(* IEC 61131-3 sources: vibrocore/firmware/codesys, 8 files *)

(* ---- GVL_IO.st ---- *)
(*
 * GVL_IO — Global Variable List: Physical I/O Mapping
 *
 * WAGO PFC200 XTR (750-8212) + I/O Modules:
 *   Slot 1: 750-430 XTR  — 4× Digital Input  24V DC  → %IX0.0..%IX0.3
 *   Slot 2: 750-530 XTR  — 4× Digital Output 24V DC  → %QX0.0..%QX0.3
 *   Slot 3: 750-637      — Incremental Encoder        → %IW4 (32-bit via IW4+IW5)
 *   Slot 4: 750-826      — RS-485 Modbus RTU          → COM config in hardware tree
 *   Slot 5: 750-600      — End module
 *
 * RS-485 Slave Addresses:
 *   Addr 1: Siemens V20 VFD  (Sonic Head)
 *   Addr 2: Nanotec C5-E     (Hub stepper driver)
 *)
VAR_GLOBAL

    (* =========================================================
       Slot 1 — 750-430 XTR: 4x Digital Input 24V DC
       ========================================================= *)

    (* Upper limit switch (NC wiring — FALSE = triggered) *)
    xLimitUp        AT %IX0.0 : BOOL;

    (* Lower limit switch (NC wiring — FALSE = triggered) *)
    xLimitDown      AT %IX0.1 : BOOL;

    (* Emergency stop mushroom button (NC — FALSE = pressed) *)
    xEStop_NC       AT %IX0.2 : BOOL;

    (* Hub driver alarm output (Nanotec C5-E ALM pin, active HIGH) *)
    xHubAlarm       AT %IX0.3 : BOOL;

    (* =========================================================
       Slot 2 — 750-530 XTR: 4x Digital Output 24V DC
       ========================================================= *)

    (* Spring-applied brake: HIGH = 24V energised = brake RELEASED *)
    xBrakeRelease   AT %QX0.0 : BOOL;

    (* Hub driver enable (Nanotec C5-E ENA pin, active HIGH) *)
    xHubEnable      AT %QX0.1 : BOOL;

    (* VFD fault reset pulse (momentary, 200ms) *)
    xVFD_Reset      AT %QX0.2 : BOOL;

    (* Spare digital output — reserved for alarm beacon / HMI *)
    xAlarmBeacon    AT %QX0.3 : BOOL;

    (* =========================================================
       Slot 3 — 750-637: Incremental Encoder
       Encoder on hub chain shaft (1000 ppr, quadrature)
       Mapped as 32-bit signed integer (IW4 = low word, IW5 = high word)
       ========================================================= *)

    iEncoderLow     AT %IW4   : INT;
    iEncoderHigh    AT %IW5   : INT;

END_VAR

(* ---- GVL_PARAMS.st ---- *)
(*
 * GVL_PARAMS — Machine Parameters and Constants
 *
 * All physical machine constants. Verify against actual hardware
 * before commissioning. Speeds and thresholds are starting values
 * for field calibration.
 *)
VAR_GLOBAL CONSTANT

    (* =========================================================
       Hub Kinematics
       NEMA 42 + Neugart PLPE120-040 (40:1) + 10B-2 chain + 15T sprocket
       ========================================================= *)

    (* Encoder pulses per mm of carriage travel
       = (pulses/rev × gear_ratio) / (sprocket_teeth × chain_pitch)
       = (1000 × 4 × 40) / (15 × 15.875) = 160000 / 238.125 ≈ 671.9 *)
    rENCODER_PULSES_PER_MM  : REAL := 671.9;

    (* Maximum carriage travel (mm) — physical mast stroke *)
    rMAX_STROKE_MM          : REAL := 1300.0;

    (* Default sampling target depth (mm from home) *)
    rTARGET_DEPTH_MM        : REAL := 1200.0;

    (* Hub speed setpoints (mm/s) *)
    rSPEED_PENETRATE_MMS    : REAL := 15.0;   (* push-in with sonic active *)
    rSPEED_RETRACT_MMS      : REAL := 50.0;   (* pull-out after sonic stop *)
    rSPEED_MANUAL_MMS       : REAL := 30.0;   (* manual jog speed *)
    rSPEED_HOMING_MMS       : REAL := 40.0;   (* homing to upper limit *)

    (* Position tolerance for "at target" check (mm) *)
    rPOS_TOLERANCE_MM       : REAL := 5.0;

    (* =========================================================
       Hub Modbus (Nanotec C5-E — CiA 402 via Modbus RTU)
       ========================================================= *)

    iHUB_SLAVE_ADDR         : INT  := 2;

    (* Modbus register addresses (holding registers, 0-based Modbus) *)
    iHUB_REG_CONTROLWORD    : INT  := 16#6040;  (* CiA 402 control word *)
    iHUB_REG_STATUSWORD     : INT  := 16#6041;  (* CiA 402 status word *)
    iHUB_REG_TARGET_VEL     : INT  := 16#60FF;  (* target velocity, rpm *)
    iHUB_REG_ACTUAL_POS     : INT  := 16#6064;  (* position actual, encoder counts *)
    iHUB_REG_OPMODE         : INT  := 16#6060;  (* modes of operation: 3=Velocity *)

    (* CiA 402 control words *)
    wHUB_CW_SHUTDOWN        : WORD := 16#0006;  (* Shutdown *)
    wHUB_CW_ENABLE          : WORD := 16#000F;  (* Switch On + Enable Op *)
    wHUB_CW_QUICKSTOP       : WORD := 16#000B;  (* Quick stop *)
    wHUB_CW_FAULT_RESET     : WORD := 16#0080;  (* Fault reset *)

    (* =========================================================
       VFD Modbus (Siemens V20 — USS/Modbus profile)
       Standard parameter channel + process data (PKW + PZD)
       ========================================================= *)

    iVFD_SLAVE_ADDR         : INT  := 1;

    (* Process data input/output word addresses (0-based) *)
    iVFD_REG_CONTROL        : INT  := 100;   (* STW1: control word *)
    iVFD_REG_FREQ_SP        : INT  := 101;   (* HSW: freq setpoint ×100 Hz *)
    iVFD_REG_STATUS         : INT  := 110;   (* ZSW1: status word *)
    iVFD_REG_FREQ_ACT       : INT  := 111;   (* HIW: actual frequency ×100 Hz *)
    iVFD_REG_CURRENT        : INT  := 112;   (* actual current ×10 A *)

    (* V20 STW1 control words *)
    wVFD_CW_START           : WORD := 16#047F;  (* bits: ON + no OFF2 + no OFF3 + OpEnable *)
    wVFD_CW_STOP_NORMAL     : WORD := 16#047E;  (* OFF1: ramp down via P1121 *)
    wVFD_CW_STOP_FAST       : WORD := 16#047B;  (* OFF3: fast ramp via P1135 + DC brake *)
    wVFD_CW_FAULT_RESET     : WORD := 16#04FE;  (* fault acknowledgement *)

    (* Frequency limits (Hz) *)
    rVFD_FREQ_MIN_HZ        : REAL := 30.0;
    rVFD_FREQ_MAX_HZ        : REAL := 110.0;
    rVFD_FREQ_DEFAULT_HZ    : REAL := 100.0;

    (* Ramp rates for software-side tracking (Hz per 100ms cycle) *)
    rVFD_RAMP_UP_HZ_STEP    : REAL := 1.5;   (* ≈15 Hz/s -->  ~7s to 100 Hz *)
    rVFD_RAMP_DN_HZ_STEP    : REAL := 4.5;   (* ≈45 Hz/s --> normal stop *)

    (* Skip resonance band: avoid 8–25 Hz during run-up *)
    rVFD_SKIP_BAND_LOW_HZ   : REAL := 8.0;
    rVFD_SKIP_BAND_HIGH_HZ  : REAL := 25.0;

    (* =========================================================
       Safety / Stone Detection
       ========================================================= *)

    (* VFD output current threshold for stone detection (% of motor rated) *)
    rSTONE_CURRENT_PCT_THR  : REAL := 130.0;

    (* Debounce time before stone alarm is confirmed *)
    tSTONE_DEBOUNCE         : TIME := T#250MS;

    (* Hub retract distance after stone detection (mm) *)
    rSTONE_RETRACT_MM       : REAL := 50.0;

    (* Max wait time for Sonic head to confirm stop before fault *)
    tSONIC_STOP_TIMEOUT     : TIME := T#5S;

    (* =========================================================
       Data / Identity
       ========================================================= *)

    sMACHINE_ID             : STRING[20] := 'VIBROCORE-001';
    sHARDWARE_VERSION       : STRING[10] := 'V1.0';
    sFIRMWARE_VERSION       : STRING[10] := '1.0.0';

END_VAR

(* ---- FB_DataLogger.st ---- *)
(*
 * FB_DataLogger — Cycle Data Logging and MQTT Payload Builder
 *
 * On each completed sampling cycle, assembles a JSON payload containing:
 *   - Machine ID, cycle number, timestamp
 *   - GPS coordinates (received from SE050/ESP32-C3 via UART → Modbus)
 *   - Achieved depth, VFD frequency, motor current
 *   - sign_pending flag → ESP32-C3 picks this up and signs via SE050 (secp256k1)
 *     then publishes to RDDL/Planetmint for VM0042 data provenance
 *
 * UART connection ESP32-C3 (RDDL Trust Wallet):
 *   WAGO COM1 (750-650 or PFC onboard UART) ↔ ESP32-C3 TX/RX
 *   Protocol: simple JSON lines at 115200 baud
 *   ESP32-C3 pushes GPS fixes every 1s: {"lat":47.123,"lon":16.456,"fix":"RTK"}
 *   WAGO sends completed cycle JSON: {"machine_id":...,"sign_pending":true}
 *   ESP32-C3 signs with SE050 and forwards to RDDL
 *
 * MQTT (WAGO onboard MQTT client via e!COCKPIT or Node-RED on PFC Linux):
 *   Topic: vibrocore/{machine_id}/cycles
 *   Broker: configured in WAGO web interface (wago-mqtt-config)
 *)
FUNCTION_BLOCK FB_DataLogger
VAR_INPUT
    xCycleTrigger       : BOOL;   (* rising edge = new cycle to log *)
    rDepth_mm           : REAL;
    rFreq_Hz            : REAL;
    rCurrent_A          : REAL;
    iSafetyReason       : INT;    (* 0=normal, >0 = what caused stop *)
END_VAR

VAR_OUTPUT
    sJSON_Payload       : STRING[500];
    xNewPayload         : BOOL;   (* TRUE for one PLC cycle when payload ready *)
    iCycleCount         : INT;
END_VAR

VAR
    (* GPS data received from ESP32-C3 — updated via UART parse task *)
    rGPS_Lat            : REAL := 0.0;
    rGPS_Lon            : REAL := 0.0;
    sGPS_Fix            : STRING[10] := 'NONE';

    tTimestamp          : TON;   (* simple uptime counter in seconds *)
    iUptimeSec          : DINT  := 0;

    xTriggerEdge        : R_TRIG;
    xPayloadSent        : BOOL;
END_VAR

(* ---- Uptime counter ---- *)
tTimestamp(IN := TRUE, PT := T#1S);
IF tTimestamp.Q THEN
    tTimestamp(IN := FALSE);
    iUptimeSec := iUptimeSec + 1;
END_IF;

(* ---- Rising edge on cycle trigger ---- *)
xTriggerEdge(CLK := xCycleTrigger);
xNewPayload := FALSE;

IF xTriggerEdge.Q THEN
    iCycleCount := iCycleCount + 1;

    (*
     * Build JSON payload manually (no dynamic allocator in IEC 61131-3).
     * Payload is read by the ESP32-C3 on COM1. The ESP32-C3 appends the
     * SE050 secp256k1 signature and publishes to RDDL/Planetmint.
     *
     * Example output:
     * {"machine_id":"VIBROCORE-001","fw":"1.0.0","cycle":1,
     *  "uptime_s":3600,"depth_mm":1198.4,"freq_hz":100.0,
     *  "current_a":1.38,"stop_reason":0,
     *  "lat":47.1234567,"lon":16.4567890,"fix":"RTK",
     *  "sign_pending":true}
     *)
    sJSON_Payload := CONCAT('{"machine_id":"',
                     CONCAT(GVL_PARAMS.sMACHINE_ID,         '","'));
    sJSON_Payload := CONCAT(sJSON_Payload,
                     CONCAT('fw":"',
                     CONCAT(GVL_PARAMS.sFIRMWARE_VERSION,   '",')));
    sJSON_Payload := CONCAT(sJSON_Payload,
                     CONCAT('"cycle":',
                     CONCAT(INT_TO_STRING(iCycleCount),     ',')));
    sJSON_Payload := CONCAT(sJSON_Payload,
                     CONCAT('"uptime_s":',
                     CONCAT(DINT_TO_STRING(iUptimeSec),     ',')));
    sJSON_Payload := CONCAT(sJSON_Payload,
                     CONCAT('"depth_mm":',
                     CONCAT(REAL_TO_STRING(rDepth_mm),      ',')));
    sJSON_Payload := CONCAT(sJSON_Payload,
                     CONCAT('"freq_hz":',
                     CONCAT(REAL_TO_STRING(rFreq_Hz),       ',')));
    sJSON_Payload := CONCAT(sJSON_Payload,
                     CONCAT('"current_a":',
                     CONCAT(REAL_TO_STRING(rCurrent_A),     ',')));
    sJSON_Payload := CONCAT(sJSON_Payload,
                     CONCAT('"stop_reason":',
                     CONCAT(INT_TO_STRING(iSafetyReason),   ',')));
    sJSON_Payload := CONCAT(sJSON_Payload,
                     CONCAT('"lat":',
                     CONCAT(REAL_TO_STRING(rGPS_Lat),       ',')));
    sJSON_Payload := CONCAT(sJSON_Payload,
                     CONCAT('"lon":',
                     CONCAT(REAL_TO_STRING(rGPS_Lon),       ',')));
    sJSON_Payload := CONCAT(sJSON_Payload,
                     CONCAT('"fix":"',
                     CONCAT(sGPS_Fix,                       '",')));
    sJSON_Payload := CONCAT(sJSON_Payload, '"sign_pending":true}');

    xNewPayload := TRUE;
END_IF;

(* ---- FB_HubControl.st ---- *)
(*
 * FB_HubControl — Hub Lift/Lower State Machine
 *
 * Controls NEMA 42 stepper via Nanotec C5-E (Modbus RTU, CiA 402).
 * Drive train: NEMA42 → Neugart PLPE120-040 (40:1) → 10B-2 chain → carriage.
 *
 * CRITICAL INTERLOCK:
 *   Hub may ONLY move upward (retract) when xSonicConfirmedStopped = TRUE.
 *   This prevents soil sample falling out during extraction.
 *   Stone detection also requires sonic stop FIRST — never retract while vibrating.
 *
 * State machine:
 *   0 IDLE          — brake engaged, motor disabled
 *   1 HOMING        — move up until xLimitUp (establishes position zero)
 *   2 DRILL_WAIT    — waiting for sonic confirmed running before hub moves
 *   3 DRILLING      — hub moves down at penetration speed
 *   4 STOP_SONIC    — target/stone reached: brake hub, request sonic fast-stop
 *   5 RETRACT       — sonic confirmed stopped, hub moves up
 *   6 ESTOP_HOLD    — emergency stop: brake engaged, waiting for release
 *   7 FAULT         — driver alarm or timeout
 *)
FUNCTION_BLOCK FB_HubControl
VAR_INPUT
    xEnable                 : BOOL;
    xSafeState              : BOOL;   (* from FB_Safety: freeze all motion *)
    xStoneDetected          : BOOL;   (* from FB_Safety: obstacle detected *)
    xSonicRunning           : BOOL;   (* from FB_SonicHead: motors spinning *)
    xSonicConfirmedStopped  : BOOL;   (* from FB_SonicHead: motors confirmed at rest *)

    rTargetDepth_mm         : REAL;   (* sampling target depth (mm from home) *)

    (* Manual jog inputs (active only in IDLE state) *)
    xCmdJogDown             : BOOL;
    xCmdJogUp               : BOOL;

    (* Auto cycle start *)
    xCmdCycleStart          : BOOL;

    (* Fault reset *)
    xCmdReset               : BOOL;
END_VAR

VAR_OUTPUT
    rPosition_mm        : REAL;    (* current carriage position from home, mm *)
    xAtHome             : BOOL;    (* carriage at upper limit *)
    xAtTarget           : BOOL;    (* carriage within tolerance of target depth *)
    xNeedSonicStop      : BOOL;    (* TRUE = request sonic fast-stop *)
    xCycleComplete      : BOOL;    (* pulse: TRUE for one cycle after retract done *)
    xFault              : BOOL;
    eState              : INT;

    (* Physical outputs — mapped by PRG_Main to GVL_IO *)
    xBrakeRelease_out   : BOOL;
    xHubEnable_out      : BOOL;
END_VAR

VAR
    (* Modbus to Nanotec C5-E *)
    fbMBWrite           : WagoModbusMasterRtu.MB_RTU_WRITE_REGS;
    fbMBRead            : WagoModbusMasterRtu.MB_RTU_READ_REGS;
    awWriteRegs         : ARRAY[0..1] OF WORD;   (* controlword + target velocity *)
    awReadRegs          : ARRAY[0..2] OF WORD;   (* statusword + actual pos low/high *)

    tMBCycle            : TON;
    tSonicStopTimeout   : TON;
    tCyclePulse         : TON;

    iSpeedSetpoint_rpm  : INT;   (* speed sent to C5-E, signed: + = down, - = up *)
    wHubCtrlWord        : WORD;

    (* 32-bit encoder position from Modbus *)
    lActualPos          : LINT;
    iPosPrev            : INT;
END_VAR

(* ---- Position calculation (encoder → mm) ---- *)
(* Combine low and high words from C5-E position register *)
lActualPos   := SHL(LINT#0 + INT_TO_LINT(awReadRegs[2]), 16)
                + INT_TO_LINT(WORD_TO_INT(awReadRegs[1]));
rPosition_mm := LINT_TO_REAL(lActualPos) / GVL_PARAMS.rENCODER_PULSES_PER_MM;

(* ---- Derived position flags ---- *)
xAtHome   := NOT GVL_IO.xLimitUp_NC;   (* NC: FALSE = triggered = home *)
xAtTarget := (rPosition_mm >= rTargetDepth_mm - GVL_PARAMS.rPOS_TOLERANCE_MM)
          AND (rPosition_mm <= rTargetDepth_mm + GVL_PARAMS.rPOS_TOLERANCE_MM);

(* ---- Global E-Stop / Safety override ---- *)
IF xSafeState AND eState <> 6 AND eState <> 7 THEN
    wHubCtrlWord        := GVL_PARAMS.wHUB_CW_QUICKSTOP;
    iSpeedSetpoint_rpm  := 0;
    xBrakeRelease_out   := FALSE;   (* brake engages *)
    xHubEnable_out      := FALSE;
    xNeedSonicStop      := TRUE;
    eState              := 6;
END_IF;

(* ---- State machine ---- *)
CASE eState OF

    (* ============================================================ *)
    0: (* IDLE *)
    (* ============================================================ *)
        wHubCtrlWord       := GVL_PARAMS.wHUB_CW_SHUTDOWN;
        iSpeedSetpoint_rpm := 0;
        xBrakeRelease_out  := FALSE;
        xHubEnable_out     := FALSE;
        xNeedSonicStop     := FALSE;
        xFault             := FALSE;
        xCyclePulse(IN := FALSE);

        IF xCmdCycleStart AND xEnable AND NOT xSafeState THEN
            eState := 1;   (* Home first, then drill *)
        ELSIF xCmdJogDown AND xEnable AND NOT GVL_IO.xLimitDown AND NOT xSafeState THEN
            xBrakeRelease_out  := TRUE;
            xHubEnable_out     := TRUE;
            wHubCtrlWord       := GVL_PARAMS.wHUB_CW_ENABLE;
            iSpeedSetpoint_rpm := REAL_TO_INT(GVL_PARAMS.rSPEED_MANUAL_MMS
                                              * GVL_PARAMS.rENCODER_PULSES_PER_MM / 1000.0 * 60.0);
        ELSIF xCmdJogUp AND xEnable AND NOT GVL_IO.xLimitUp AND NOT xSafeState THEN
            xBrakeRelease_out  := TRUE;
            xHubEnable_out     := TRUE;
            wHubCtrlWord       := GVL_PARAMS.wHUB_CW_ENABLE;
            iSpeedSetpoint_rpm := -REAL_TO_INT(GVL_PARAMS.rSPEED_MANUAL_MMS
                                               * GVL_PARAMS.rENCODER_PULSES_PER_MM / 1000.0 * 60.0);
        END_IF;

    (* ============================================================ *)
    1: (* HOMING — move up to upper limit switch *)
    (* ============================================================ *)
        xBrakeRelease_out  := TRUE;
        xHubEnable_out     := TRUE;
        wHubCtrlWord       := GVL_PARAMS.wHUB_CW_ENABLE;
        iSpeedSetpoint_rpm := -REAL_TO_INT(GVL_PARAMS.rSPEED_HOMING_MMS
                                           * GVL_PARAMS.rENCODER_PULSES_PER_MM / 1000.0 * 60.0);

        IF xAtHome THEN
            (* Limit reached — stop motor, set position origin in C5-E *)
            wHubCtrlWord       := GVL_PARAMS.wHUB_CW_SHUTDOWN;
            iSpeedSetpoint_rpm := 0;
            xBrakeRelease_out  := FALSE;
            xHubEnable_out     := FALSE;
            eState             := 2;   (* → wait for sonic *)
        END_IF;

    (* ============================================================ *)
    2: (* DRILL_WAIT — wait for sonic confirmed running *)
    (* ============================================================ *)
        xBrakeRelease_out  := FALSE;
        xHubEnable_out     := FALSE;
        iSpeedSetpoint_rpm := 0;

        IF xSonicRunning THEN
            eState := 3;
        END_IF;

        IF NOT xEnable OR xSafeState THEN
            eState := 0;
        END_IF;

    (* ============================================================ *)
    3: (* DRILLING — hub moves down, sonic running *)
    (* ============================================================ *)
        xBrakeRelease_out  := TRUE;
        xHubEnable_out     := TRUE;
        wHubCtrlWord       := GVL_PARAMS.wHUB_CW_ENABLE;
        iSpeedSetpoint_rpm := REAL_TO_INT(GVL_PARAMS.rSPEED_PENETRATE_MMS
                                          * GVL_PARAMS.rENCODER_PULSES_PER_MM / 1000.0 * 60.0);

        (* Stop drilling on target OR stone *)
        IF xAtTarget OR xStoneDetected OR GVL_IO.xLimitDown THEN
            (* Engage brake, request sonic fast-stop *)
            wHubCtrlWord       := GVL_PARAMS.wHUB_CW_QUICKSTOP;
            iSpeedSetpoint_rpm := 0;
            xBrakeRelease_out  := FALSE;
            xHubEnable_out     := FALSE;
            xNeedSonicStop     := TRUE;
            eState             := 4;
        END_IF;

    (* ============================================================ *)
    4: (* STOP_SONIC — brake engaged, waiting for sonic to confirm stop *)
    (* Hub MUST NOT move. Retract only after xSonicConfirmedStopped. *)
    (* ============================================================ *)
        xBrakeRelease_out  := FALSE;
        xHubEnable_out     := FALSE;
        iSpeedSetpoint_rpm := 0;
        xNeedSonicStop     := TRUE;   (* keep requesting fast stop *)

        tSonicStopTimeout(
            IN := TRUE,
            PT := GVL_PARAMS.tSONIC_STOP_TIMEOUT
        );

        IF xSonicConfirmedStopped THEN
            tSonicStopTimeout(IN := FALSE);
            xNeedSonicStop := FALSE;
            eState := 5;   (* → now safe to retract *)
        END_IF;

        IF tSonicStopTimeout.Q THEN
            tSonicStopTimeout(IN := FALSE);
            xFault := TRUE;
            eState := 7;   (* timeout waiting for sonic → fault *)
        END_IF;

    (* ============================================================ *)
    5: (* RETRACT — sonic confirmed stopped, hub moves up *)
    (* ============================================================ *)
        xBrakeRelease_out  := TRUE;
        xHubEnable_out     := TRUE;
        wHubCtrlWord       := GVL_PARAMS.wHUB_CW_ENABLE;
        iSpeedSetpoint_rpm := -REAL_TO_INT(GVL_PARAMS.rSPEED_RETRACT_MMS
                                           * GVL_PARAMS.rENCODER_PULSES_PER_MM / 1000.0 * 60.0);

        IF xAtHome THEN
            wHubCtrlWord       := GVL_PARAMS.wHUB_CW_SHUTDOWN;
            iSpeedSetpoint_rpm := 0;
            xBrakeRelease_out  := FALSE;
            xHubEnable_out     := FALSE;
            (* Pulse xCycleComplete for one cycle *)
            tCyclePulse(IN := TRUE, PT := T#500MS);
            xCycleComplete     := tCyclePulse.Q;
            IF tCyclePulse.Q THEN
                tCyclePulse(IN := FALSE);
                xCycleComplete := FALSE;
                eState := 0;
            END_IF;
        END_IF;

    (* ============================================================ *)
    6: (* ESTOP_HOLD — hold until E-Stop released and reset *)
    (* ============================================================ *)
        wHubCtrlWord       := GVL_PARAMS.wHUB_CW_QUICKSTOP;
        iSpeedSetpoint_rpm := 0;
        xBrakeRelease_out  := FALSE;
        xHubEnable_out     := FALSE;
        xNeedSonicStop     := TRUE;

        IF NOT xSafeState AND xCmdReset THEN
            xNeedSonicStop := FALSE;
            eState := 1;   (* Re-home after E-Stop *)
        END_IF;

    (* ============================================================ *)
    7: (* FAULT — driver alarm or sonic stop timeout *)
    (* ============================================================ *)
        wHubCtrlWord       := GVL_PARAMS.wHUB_CW_QUICKSTOP;
        iSpeedSetpoint_rpm := 0;
        xBrakeRelease_out  := FALSE;
        xHubEnable_out     := FALSE;
        xFault             := TRUE;

        IF xCmdReset AND NOT xSafeState AND NOT GVL_IO.xHubAlarm THEN
            xFault := FALSE;
            eState := 0;
        END_IF;

END_CASE;

(* ---- Nanotec C5-E Modbus write (20ms cycle) ---- *)
tMBCycle(IN := NOT tMBCycle.Q, PT := T#20MS);
IF tMBCycle.Q THEN
    awWriteRegs[0] := wHubCtrlWord;
    awWriteRegs[1] := INT_TO_WORD(iSpeedSetpoint_rpm);

    fbMBWrite(
        bExecute      := TRUE,
        nSlaveAddress := BYTE#2,
        eFunction     := WagoModbusMasterRtu.eMBFC.WriteMultipleRegisters,
        nStartAddress := INT_TO_WORD(GVL_PARAMS.iHUB_REG_CONTROLWORD),
        nQuantity     := 2,
        pData         := ADR(awWriteRegs),
        nDataLen      := SIZEOF(awWriteRegs)
    );

    fbMBRead(
        bExecute      := TRUE,
        nSlaveAddress := BYTE#2,
        eFunction     := WagoModbusMasterRtu.eMBFC.ReadHoldingRegisters,
        nStartAddress := INT_TO_WORD(GVL_PARAMS.iHUB_REG_STATUSWORD),
        nQuantity     := 3,
        pData         := ADR(awReadRegs),
        nDataLen      := SIZEOF(awReadRegs)
    );
END_IF;

(* ---- FB_ModbusVFD.st ---- *)
(*
 * FB_ModbusVFD — Siemens V20 VFD Communication via Modbus RTU
 *
 * Hardware: WAGO 750-826 RS-485 module, COM2 port
 * VFD: Siemens SINAMICS V20, Modbus slave address 1
 *
 * V20 pre-commissioning (set via BOP or STARTER):
 *   P0700 = 5     (command source: Modbus)
 *   P1000 = 5     (freq setpoint: Modbus)
 *   P2010[0] = 6  (Modbus baud: 9600)
 *   P2011[0] = 1  (slave address: 1)
 *   P2012[0] = 2  (PZD word count: 2)
 *   P1120 = 5.0   (ramp-up time, s)
 *   P1121 = 3.0   (ramp-down time OFF1, s)
 *   P1135 = 0.3   (ramp-down time OFF3 fast-stop, s)
 *   P1232 = 100   (DC braking current %)
 *   P1233 = 0.5   (DC braking duration, s)
 *
 * Control word bits (STW1):
 *   Bit 0: ON/OFF1  (0 = ramp to stop via P1121)
 *   Bit 1: no OFF2  (0 = coast to stop — keep 1)
 *   Bit 2: no OFF3  (0 = fast stop via P1135 — used for fast stop)
 *   Bit 3: enable operation
 *   Bit 6: setpoint enable
 *   Bit 7: fault acknowledge
 *
 * Note: Modbus library used is WagoAppModbusMasterRtu (WAGO CODESYS package).
 * Import via Library Manager: WagoAppModbusMasterRtu >= 1.1.0.0
 *)
FUNCTION_BLOCK FB_ModbusVFD
VAR_INPUT
    xEnable         : BOOL;   (* FALSE = VFD disabled, no communication *)
    xStart          : BOOL;   (* TRUE = run motor *)
    xFastStop       : BOOL;   (* TRUE = OFF3 immediately (stone / safety) *)
    xFaultReset     : BOOL;   (* rising edge = reset VFD fault *)
    rFreqSetpoint   : REAL;   (* Hz, clamped internally to MIN/MAX *)
END_VAR

VAR_OUTPUT
    xRunning        : BOOL;   (* TRUE = VFD reports motor running *)
    xReady          : BOOL;   (* TRUE = VFD ready for start command *)
    xFault          : BOOL;   (* TRUE = VFD in fault state *)
    rFreqActual     : REAL;   (* Hz — actual output frequency *)
    rCurrentActual  : REAL;   (* A  — actual output current *)
    rCurrent_pct    : REAL;   (* % of motor rated current (rated = 1.45A) *)
    xCommError      : BOOL;   (* TRUE = Modbus communication lost *)
END_VAR

VAR
    (* Modbus master FB — WagoAppModbusMasterRtu library *)
    fbMBWrite       : WagoModbusMasterRtu.MB_RTU_WRITE_REGS;
    fbMBRead        : WagoModbusMasterRtu.MB_RTU_READ_REGS;

    awWriteRegs     : ARRAY[0..1] OF WORD;   (* control + freq setpoint *)
    awReadRegs      : ARRAY[0..2] OF WORD;   (* status + freq actual + current *)

    wControlWord    : WORD;
    iFreqRaw        : INT;

    tCycle          : TON;     (* 20ms poll cycle *)
    tCommTimeout    : TON;     (* Modbus comms watchdog *)

    xResetEdge      : R_TRIG;
    xLastFaultReset : BOOL;

    (* Motor rated current for % calculation — OLI MVE 400/6-HF: 1.45A at 230V 3ph *)
    rRATED_CURRENT  : REAL := 1.45;
END_VAR

(* ---- Fault reset edge detection ---- *)
xResetEdge(CLK := xFaultReset);

(* ---- Build control word ---- *)
IF NOT xEnable THEN
    wControlWord := 16#0000;   (* fully disabled *)

ELSIF xFastStop THEN
    (* OFF3: bit 2 = 0 → VFD uses P1135 ramp + DC brake *)
    (* Achieves motor stop in ~200–400ms (vs 3+ s for normal ramp) *)
    wControlWord := GVL_PARAMS.wVFD_CW_STOP_FAST;

ELSIF xResetEdge.Q THEN
    wControlWord := GVL_PARAMS.wVFD_CW_FAULT_RESET;

ELSIF xStart THEN
    wControlWord := GVL_PARAMS.wVFD_CW_START;

ELSE
    (* Normal stop: OFF1, ramps down via P1121 *)
    wControlWord := GVL_PARAMS.wVFD_CW_STOP_NORMAL;
END_IF;

(* ---- Frequency setpoint (V20: value = Hz × 100) ---- *)
iFreqRaw := REAL_TO_INT(
    MAX(GVL_PARAMS.rVFD_FREQ_MIN_HZ,
        MIN(GVL_PARAMS.rVFD_FREQ_MAX_HZ, rFreqSetpoint)) * 100.0
);

(* ---- Pack write registers ---- *)
awWriteRegs[0] := wControlWord;
awWriteRegs[1] := INT_TO_WORD(iFreqRaw);

(* ---- 20ms poll cycle ---- *)
tCycle(IN := NOT tCycle.Q, PT := T#20MS);

IF tCycle.Q AND xEnable THEN

    (* Write: control word + freq setpoint *)
    fbMBWrite(
        bExecute     := TRUE,
        nSlaveAddress := BYTE#1,
        eFunction    := WagoModbusMasterRtu.eMBFC.WriteMultipleRegisters,
        nStartAddress := INT_TO_WORD(GVL_PARAMS.iVFD_REG_CONTROL),
        nQuantity    := 2,
        pData        := ADR(awWriteRegs),
        nDataLen     := SIZEOF(awWriteRegs)
    );

    (* Read: status word + actual freq + actual current *)
    fbMBRead(
        bExecute     := TRUE,
        nSlaveAddress := BYTE#1,
        eFunction    := WagoModbusMasterRtu.eMBFC.ReadHoldingRegisters,
        nStartAddress := INT_TO_WORD(GVL_PARAMS.iVFD_REG_STATUS),
        nQuantity    := 3,
        pData        := ADR(awReadRegs),
        nDataLen     := SIZEOF(awReadRegs)
    );

    IF fbMBRead.bDone AND NOT fbMBRead.bError THEN
        xCommError  := FALSE;
        (* ZSW1 status word bits *)
        xReady      := awReadRegs[0].1;   (* Bit 1: ready to switch on *)
        xRunning    := awReadRegs[0].2;   (* Bit 2: operation enabled / running *)
        xFault      := awReadRegs[0].3;   (* Bit 3: fault *)
        rFreqActual := WORD_TO_INT(awReadRegs[1]) / 100.0;
        rCurrentActual := WORD_TO_INT(awReadRegs[2]) / 10.0;
        rCurrent_pct   := (rCurrentActual / rRATED_CURRENT) * 100.0;
        tCommTimeout(IN := FALSE);
    ELSE
        tCommTimeout(IN := TRUE, PT := T#2S);
        xCommError := tCommTimeout.Q;
    END_IF;

END_IF;

(* ---- FB_Safety.st ---- *)
(*
 * FB_Safety — Safety Monitor Function Block
 *
 * Evaluates all safety-relevant inputs and sets xSafeState.
 * When xSafeState = TRUE, all motion must stop immediately.
 *
 * Safety categories addressed:
 *   - E-Stop: Category 3 (redundant NC wiring evaluated here)
 *   - Limit switches: NC wiring, software evaluation
 *   - Overcurrent / stone detection: software function
 *   - Hub driver fault: hardware alarm signal
 *   - VFD fault: reported by FB_ModbusVFD
 *
 * IMPORTANT: This FB does NOT directly cut power. Physical power cut
 * is handled by the safety relay (Pilz PNOZ or equivalent) wired in
 * series with the 24V supply to the VFD enable and brake circuit.
 * This FB provides the software-level interlock for the state machines.
 *)
FUNCTION_BLOCK FB_Safety
VAR_INPUT
    (* E-Stop NC contact — FALSE when button pressed *)
    xEStop_NC           : BOOL;

    (* Limit switches — NC wiring, FALSE = triggered *)
    xLimitUp_NC         : BOOL;
    xLimitDown_NC       : BOOL;

    (* Hub driver alarm output (active HIGH) *)
    xHubAlarm           : BOOL;

    (* VFD fault flag from FB_ModbusVFD *)
    xVFD_Fault          : BOOL;

    (* VFD output current as percentage of motor rated current
       Provided by FB_ModbusVFD after scaling *)
    rVFD_Current_pct    : REAL;

    (* Current hub movement direction (TRUE = moving down) *)
    xHubMovingDown      : BOOL;

    (* Current hub movement direction (TRUE = moving up) *)
    xHubMovingUp        : BOOL;
END_VAR

VAR_OUTPUT
    (* TRUE = safe state active — all motion must stop *)
    xSafeState          : BOOL;

    (* TRUE = stone/obstacle detected during penetration *)
    xStoneDetected      : BOOL;

    (* Upper limit triggered (only blocks upward movement) *)
    xLimitUpTriggered   : BOOL;

    (* Lower limit triggered (only blocks downward movement) *)
    xLimitDownTriggered : BOOL;

    (* Reason code: 0=OK 1=EStop 2=HubAlarm 3=VFD 4=Stone *)
    eSafetyReason       : INT;
END_VAR

VAR
    tStoneDebounce      : TON;
END_VAR

(* ---- Limit switch evaluation (NC contacts: FALSE = triggered) ---- *)
xLimitUpTriggered   := NOT xLimitUp_NC;
xLimitDownTriggered := NOT xLimitDown_NC;

(* ---- Stone detection with debounce ---- *)
tStoneDebounce(
    IN := rVFD_Current_pct > GVL_PARAMS.rSTONE_CURRENT_PCT_THR,
    PT := GVL_PARAMS.tSTONE_DEBOUNCE
);
xStoneDetected := tStoneDebounce.Q;

(* ---- Safe state evaluation (priority order) ---- *)
xSafeState    := FALSE;
eSafetyReason := 0;

IF NOT xEStop_NC THEN
    (* E-Stop has highest priority — hard stop *)
    xSafeState    := TRUE;
    eSafetyReason := 1;

ELSIF xHubAlarm THEN
    (* Hub driver hardware fault *)
    xSafeState    := TRUE;
    eSafetyReason := 2;

ELSIF xVFD_Fault THEN
    (* VFD hardware fault *)
    xSafeState    := TRUE;
    eSafetyReason := 3;

ELSIF xStoneDetected THEN
    (* Overcurrent → stone/obstacle — handled by state machine,
       but also sets safe state to freeze motion *)
    xSafeState    := TRUE;
    eSafetyReason := 4;

ELSIF xLimitUpTriggered AND xHubMovingUp THEN
    (* Limit in direction of travel — stop motion *)
    xSafeState    := TRUE;
    eSafetyReason := 5;

ELSIF xLimitDownTriggered AND xHubMovingDown THEN
    (* Limit in direction of travel — stop motion *)
    xSafeState    := TRUE;
    eSafetyReason := 6;
END_IF;

(* ---- FB_SonicHead.st ---- *)
(*
 * FB_SonicHead — Sonic Head State Machine
 *
 * Controls 2× OLI MVE 400/6-HF via Siemens V20 VFD (Modbus RTU).
 * Provides adaptive frequency control based on VFD load current.
 *
 * CRITICAL STOP BEHAVIOUR:
 *   - xFastStop = TRUE  → OFF3 command to VFD immediately
 *                         VFD uses P1135 ramp (0.3s) + DC injection braking
 *                         Expected motor standstill: 200–400ms
 *   - xFastStop = FALSE → OFF1 normal ramp (P1121, 3s) for end-of-cycle stop
 *
 * State machine:
 *   0 IDLE       — VFD disabled, motors at rest
 *   1 STARTING   — VFD enabled, ramping up, skip resonance band
 *   2 RUNNING    — Full speed, adaptive freq control active
 *   3 STOPPING   — Normal OFF1 stop (end of cycle)
 *   4 FAST_STOP  — OFF3 stop (stone / safety / E-Stop)
 *   5 FAULT      — VFD or comms fault, waits for reset
 *
 * Output xConfirmedStopped = TRUE only when VFD reports NOT running
 * AND state machine is in IDLE. Hub retract must wait for this.
 *)
FUNCTION_BLOCK FB_SonicHead
VAR_INPUT
    xEnable         : BOOL;   (* Allow sonic head to run *)
    xSafeState      : BOOL;   (* Safety FB active → fast stop *)
    xFastStop       : BOOL;   (* External fast stop request (stone, end-of-cycle) *)
    rTargetFreq_Hz  : REAL;   (* Desired operating frequency 30–110 Hz *)
    xFaultReset     : BOOL;   (* Reset VFD fault *)
END_VAR

VAR_OUTPUT
    xRunning            : BOOL;   (* TRUE = OLI motors are rotating *)
    xConfirmedStopped   : BOOL;   (* TRUE = motors confirmed at standstill *)
    xFault              : BOOL;
    rActualFreq_Hz      : REAL;
    rActualCurrent_A    : REAL;
    rActualCurrent_pct  : REAL;
    eState              : INT;
END_VAR

VAR
    fbVFD               : FB_ModbusVFD;

    rCurrentFreq        : REAL  := 0.0;   (* tracked setpoint sent to VFD *)
    tRampTick           : TON;            (* 100ms ramp tick *)
    tFastStopTimeout    : TON;            (* watchdog: motor must stop within 5s *)
    tFastStopConfirm    : TON;            (* confirm standstill for 200ms *)

    xFastStopActive     : BOOL;
    xNormalStopActive   : BOOL;
END_VAR

(* ---- Resolve stop type ---- *)
xFastStopActive   := xFastStop OR xSafeState;
xNormalStopActive := (NOT xEnable) AND (NOT xFastStopActive);

(* ---- State machine ---- *)
CASE eState OF

    (* ============================================================ *)
    0: (* IDLE — motors at rest *)
    (* ============================================================ *)
        rCurrentFreq  := 0.0;
        xConfirmedStopped := NOT fbVFD.xRunning;

        IF xEnable AND NOT xSafeState AND NOT xFastStopActive THEN
            tRampTick(IN := FALSE);
            eState := 1;
        END_IF;

        IF xFaultReset AND fbVFD.xFault THEN
            eState := 5;
        END_IF;

    (* ============================================================ *)
    1: (* STARTING — ramp up to target, skip resonance band *)
    (* ============================================================ *)
        xConfirmedStopped := FALSE;

        tRampTick(IN := NOT tRampTick.Q, PT := T#100MS);
        IF tRampTick.Q THEN
            rCurrentFreq := rCurrentFreq + GVL_PARAMS.rVFD_RAMP_UP_HZ_STEP;

            (* Skip over structural resonance band (8–25 Hz) *)
            IF rCurrentFreq > GVL_PARAMS.rVFD_SKIP_BAND_LOW_HZ
            AND rCurrentFreq < GVL_PARAMS.rVFD_SKIP_BAND_HIGH_HZ THEN
                rCurrentFreq := GVL_PARAMS.rVFD_SKIP_BAND_HIGH_HZ;
            END_IF;
        END_IF;

        IF rCurrentFreq >= rTargetFreq_Hz THEN
            rCurrentFreq := rTargetFreq_Hz;
            eState := 2;
        END_IF;

        (* Abort ramp-up if stop requested *)
        IF xFastStopActive THEN
            eState := 4;
        ELSIF xNormalStopActive THEN
            eState := 3;
        END_IF;

        IF fbVFD.xFault THEN
            eState := 5;
        END_IF;

    (* ============================================================ *)
    2: (* RUNNING — adaptive frequency control *)
    (* ============================================================ *)
        xConfirmedStopped := FALSE;

        (* Adaptive frequency: increase freq when soil resistance rises,
           decrease when soil is soft (VFD current as proxy for load) *)
        IF rActualCurrent_pct > 120.0 THEN
            (* High resistance: increase frequency towards max *)
            rCurrentFreq := MIN(GVL_PARAMS.rVFD_FREQ_MAX_HZ,
                                rCurrentFreq + 0.5);
        ELSIF rActualCurrent_pct < 50.0 THEN
            (* Low load: ease back towards min to save energy *)
            rCurrentFreq := MAX(GVL_PARAMS.rVFD_FREQ_MIN_HZ,
                                rCurrentFreq - 0.5);
        ELSE
            (* Within normal band: hold at target *)
            rCurrentFreq := rTargetFreq_Hz;
        END_IF;

        IF xFastStopActive THEN
            eState := 4;
        ELSIF xNormalStopActive THEN
            eState := 3;
        END_IF;

        IF fbVFD.xFault THEN
            eState := 5;
        END_IF;

    (* ============================================================ *)
    3: (* STOPPING — normal OFF1 ramp (end-of-cycle) *)
    (* ============================================================ *)
        (* VFD handles the ramp internally via P1121.
           We track frequency to zero for display only. *)
        tRampTick(IN := NOT tRampTick.Q, PT := T#100MS);
        IF tRampTick.Q THEN
            rCurrentFreq := MAX(0.0, rCurrentFreq - GVL_PARAMS.rVFD_RAMP_DN_HZ_STEP);
        END_IF;

        IF NOT fbVFD.xRunning AND rCurrentFreq <= 0.0 THEN
            tFastStopConfirm(IN := TRUE, PT := T#200MS);
            IF tFastStopConfirm.Q THEN
                tFastStopConfirm(IN := FALSE);
                eState := 0;
            END_IF;
        END_IF;

        (* Escalate to fast stop if safety triggers during normal stop *)
        IF xFastStopActive THEN
            eState := 4;
        END_IF;

    (* ============================================================ *)
    4: (* FAST_STOP — OFF3 immediately (stone / E-Stop / safety) *)
    (* CRITICAL: Hub must NOT retract until xConfirmedStopped = TRUE *)
    (* ============================================================ *)
        rCurrentFreq := 0.0;

        (* Watchdog: if motor does not stop within timeout → fault *)
        tFastStopTimeout(
            IN := TRUE,
            PT := GVL_PARAMS.tSONIC_STOP_TIMEOUT
        );

        IF NOT fbVFD.xRunning THEN
            (* Confirm standstill for 200ms before declaring stopped *)
            tFastStopConfirm(IN := TRUE, PT := T#200MS);
            tFastStopTimeout(IN := FALSE);

            IF tFastStopConfirm.Q THEN
                tFastStopConfirm(IN := FALSE);
                xConfirmedStopped := TRUE;

                IF NOT xFastStopActive THEN
                    eState := 0;   (* Fast stop cause cleared → back to IDLE *)
                END_IF;
            END_IF;
        ELSE
            tFastStopConfirm(IN := FALSE);
            xConfirmedStopped := FALSE;
        END_IF;

        IF tFastStopTimeout.Q THEN
            tFastStopTimeout(IN := FALSE);
            eState := 5;   (* Motor refuses to stop → fault *)
        END_IF;

    (* ============================================================ *)
    5: (* FAULT *)
    (* ============================================================ *)
        rCurrentFreq      := 0.0;
        xConfirmedStopped := FALSE;

        IF xFaultReset AND NOT fbVFD.xFault THEN
            eState := 0;
        END_IF;

END_CASE;

(* ---- Drive VFD FB ---- *)
fbVFD(
    xEnable       := xEnable OR (eState > 0),
    xStart        := (eState = 1) OR (eState = 2) OR (eState = 3),
    xFastStop     := (eState = 4),
    xFaultReset   := xFaultReset,
    rFreqSetpoint := rCurrentFreq
);

(* ---- Map outputs ---- *)
xRunning           := fbVFD.xRunning;
xFault             := fbVFD.xFault OR fbVFD.xCommError;
rActualFreq_Hz     := fbVFD.rFreqActual;
rActualCurrent_A   := fbVFD.rCurrentActual;
rActualCurrent_pct := fbVFD.rCurrent_pct;

(* ---- PRG_Main.st ---- *)
(*
 * PRG_Main — Vibrocore Main Control Program
 *
 * Orchestrates all function blocks in the correct execution order:
 *   1. FB_Safety  — always first, evaluates all safety inputs
 *   2. FB_SonicHead — VFD / OLI motor control
 *   3. FB_HubControl — carriage position and chain drive
 *   4. FB_DataLogger — cycle data and MQTT/RDDL payload
 *
 * Physical I/O outputs (from GVL_IO) are assigned ONLY here,
 * never inside function blocks.
 *
 * Operating modes (eMode):
 *   0  MANUAL   — jog up/down via HMI buttons, sonic via HMI toggle
 *   1  DT325    — automatic sampling cycle with DT325 Geoprobe core barrel
 *   2  AUGER    — automatic sampling cycle with 30mm auger (future)
 *
 * Sampling cycle sequence (DT325_AUTO):
 *
 *   IDLE → [CycleStart]
 *   → SONIC_START   : enable sonic, wait xSonicRunning
 *   → DRILLING      : hub down at penetration speed
 *   → [xAtTarget OR xStoneDetected OR xLimitDown]
 *   → STOP_SONIC    : brake hub, sonic fast-stop, wait xSonicConfirmedStopped
 *   → RETRACT       : hub up at retract speed
 *   → [xAtHome]
 *   → LOG_CYCLE     : write data, signal SE050 signing
 *   → IDLE
 *
 * INTERLOCK: Hub retract BLOCKED until fbSonic.xConfirmedStopped = TRUE.
 *            No exception. Not for stone, not for normal stop.
 *)
PROGRAM PRG_Main
VAR
    fbSafety        : FB_Safety;
    fbSonic         : FB_SonicHead;
    fbHub           : FB_HubControl;
    fbLogger        : FB_DataLogger;

    (* Operating mode selection *)
    eMode           : INT := 0;   (* 0=MANUAL 1=DT325_AUTO 2=AUGER *)

    (* Sampling target (can be overridden from HMI / Modbus PLC register) *)
    rTargetDepth_mm : REAL := GVL_PARAMS.rTARGET_DEPTH_MM;
    rTargetFreq_Hz  : REAL := GVL_PARAMS.rVFD_FREQ_DEFAULT_HZ;

    (* HMI / operator inputs (write from HMI or Modbus PLC holding register) *)
    xHMI_CycleStart : BOOL;
    xHMI_JogDown    : BOOL;
    xHMI_JogUp      : BOOL;
    xHMI_SonicToggle: BOOL;
    xHMI_FaultReset : BOOL;

    (* Status outputs (readable from HMI / remote via WAGO REST API) *)
    eSystemState    : INT;    (* mirrors sampling state *)
    sSafetyStatus   : STRING[30];
    xSystemOK       : BOOL;
END_VAR

(* ================================================================
   1. SAFETY — always executed first, every scan cycle
   ================================================================ *)
fbSafety(
    xEStop_NC           := GVL_IO.xEStop_NC,
    xLimitUp_NC         := GVL_IO.xLimitUp,
    xLimitDown_NC       := GVL_IO.xLimitDown,
    xHubAlarm           := GVL_IO.xHubAlarm,
    xVFD_Fault          := fbSonic.xFault,
    rVFD_Current_pct    := fbSonic.rActualCurrent_pct,
    xHubMovingDown      := (fbHub.eState = 3),
    xHubMovingUp        := (fbHub.eState = 5) OR (fbHub.eState = 1)
);

(* ================================================================
   2. SONIC HEAD
   ================================================================ *)
fbSonic(
    xEnable         := (eMode = 1) AND (fbHub.eState = 3 OR fbHub.eState = 2)
                       OR (eMode = 0 AND xHMI_SonicToggle),
    xSafeState      := fbSafety.xSafeState,
    xFastStop       := fbHub.xNeedSonicStop OR fbSafety.xSafeState,
    rTargetFreq_Hz  := rTargetFreq_Hz,
    xFaultReset     := xHMI_FaultReset
);

(* ================================================================
   3. HUB CONTROL
   ================================================================ *)
fbHub(
    xEnable                 := NOT fbSafety.xSafeState,
    xSafeState              := fbSafety.xSafeState,
    xStoneDetected          := fbSafety.xStoneDetected,
    xSonicRunning           := fbSonic.xRunning,
    xSonicConfirmedStopped  := fbSonic.xConfirmedStopped,
    rTargetDepth_mm         := rTargetDepth_mm,
    xCmdJogDown             := xHMI_JogDown AND (eMode = 0),
    xCmdJogUp               := xHMI_JogUp   AND (eMode = 0),
    xCmdCycleStart          := xHMI_CycleStart AND (eMode = 1),
    xCmdReset               := xHMI_FaultReset
);

(* ================================================================
   4. PHYSICAL I/O ASSIGNMENT
   Write physical outputs ONLY here, never inside FBs
   ================================================================ *)
GVL_IO.xBrakeRelease := fbHub.xBrakeRelease_out AND NOT fbSafety.xSafeState;
GVL_IO.xHubEnable    := fbHub.xHubEnable_out    AND NOT fbSafety.xSafeState;
GVL_IO.xVFD_Reset    := xHMI_FaultReset;
GVL_IO.xAlarmBeacon  := fbSafety.xSafeState OR fbHub.xFault OR fbSonic.xFault;

(* ================================================================
   5. DATA LOGGER
   ================================================================ *)
fbLogger(
    xCycleTrigger   := fbHub.xCycleComplete,
    rDepth_mm       := fbHub.rPosition_mm,
    rFreq_Hz        := fbSonic.rActualFreq_Hz,
    rCurrent_A      := fbSonic.rActualCurrent_A,
    iSafetyReason   := fbSafety.eSafetyReason
);

(* ================================================================
   6. SYSTEM STATUS SUMMARY (for HMI / remote monitoring)
   ================================================================ *)
eSystemState := fbHub.eState;
xSystemOK    := NOT fbSafety.xSafeState
             AND NOT fbHub.xFault
             AND NOT fbSonic.xFault;

CASE fbSafety.eSafetyReason OF
    0: sSafetyStatus := 'OK';
    1: sSafetyStatus := 'E-STOP PRESSED';
    2: sSafetyStatus := 'HUB DRIVER ALARM';
    3: sSafetyStatus := 'VFD FAULT';
    4: sSafetyStatus := 'STONE DETECTED';
    5: sSafetyStatus := 'UPPER LIMIT HIT';
    6: sSafetyStatus := 'LOWER LIMIT HIT';
ELSE
    sSafetyStatus := 'UNKNOWN';
END_CASE;
